TEXTLIST TL_Pparmas
  1 = 'Setpoint'
  2 = 'StandbySetpoint'
  3 = 'Setpoints[1]'
  4 = 'Setpoints[2]'
  5 = 'Setpoints[3]'
  6 = 'Setpoints[4]'
  7 = 'Setpoints[5]'
  8 = 'Threshold_PP'
  9 = 'Threshold_P'
  10 = 'Threshold_M'
  11 = 'Threshold_MM'
  12 = 'Openloop_Output'
   = ''
END_TEXTLIST

(* stored: Version 1.1.0.1, ProductVersion 3.1.4020.12
   TextList TL_Pparmas: Id {23807846-1153-4a69-8b6e-8c8184816c5e} *)
